// TIA Portal project "tonzamanrolesi_ve_asiriakim kullanimi" (V18)

(* hardware
DEVICE "S7-1200 station_1"  S7-1200 Station
   slot 0: "Rack_0"  S7-1200 Rack  Rack  V1.0
   slot 1: "PLC_1"  CPU 1214C AC/DC/Rly  6ES7 214-1BG40-0XB0  V4.6
*)

// ===== PLC "PLC_1"  CPU 1214C AC/DC/Rly =====

VAR_GLOBAL   // PLC tag table "Default tag table"
   "STOP" AT %I0.0 : Bool;
   "START" AT %I0.1 : Bool;
   "AA_1" AT %I0.2 : Bool;
   "AA_2" AT %I0.3 : Bool;
   "MOTOR_1" AT %Q0.1 : Bool;
   "MOTOR__2" AT %Q0.2 : Bool;
END_VAR

// folder: System blocks/Program resources

DATA_BLOCK "T1"   // DB1
{ S7_Optimized_Access := 'TRUE' }
AUTHOR : Simatic
FAMILY : IEC
NAME : IEC_TMR
VERSION : 1.0
// stored: InstanceOfName IEC_TIMER
"IEC_TIMER"
BEGIN
END_DATA_BLOCK

DATA_BLOCK "T2"   // DB2
{ S7_Optimized_Access := 'TRUE' }
AUTHOR : Simatic
FAMILY : IEC
NAME : IEC_TMR
VERSION : 1.0
// stored: InstanceOfName IEC_TIMER
"IEC_TIMER"
BEGIN
END_DATA_BLOCK

// folder: (top level)

ORGANIZATION_BLOCK "Main"   // OB1, LAD, ProgramCycle
TITLE = "Main Program Sweep (Cycle)"
{ S7_Optimized_Access := 'TRUE' }
VERSION : 0.1
   VAR_INPUT
      Initial_Call : Bool;   // Initial call of this OB
      Remanence : Bool;   // =True, if remanent data are available
   END_VAR
   VAR_TEMP   // added for the SCL form of the ladder/FBD networks
      _w1 : Bool;
      _w2 : Bool;
   END_VAR
BEGIN

REGION Network 1
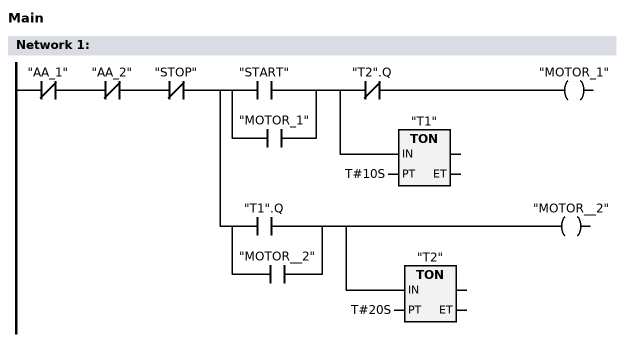
   #_w1 := NOT "AA_1" AND NOT "AA_2" AND NOT "STOP";
   #_w2 := #_w1 AND ("START" OR "MOTOR_1");
   "MOTOR_1" := #_w2 AND NOT "T2".Q;
   "T1".TON(IN := #_w2, PT := T#10S);
   "MOTOR__2" := #_w1 AND ("T1".Q OR "MOTOR__2");
   "T2".TON(IN := "MOTOR__2", PT := T#20S);
END_REGION
END_ORGANIZATION_BLOCK